INTERFACE I_Conveyor

PROPERTY bOccupied : BOOL
GET
END_GET
SET
END_SET
END_PROPERTY

PROPERTY eMode : E_ConveyorMode
GET
END_GET
SET
END_SET
END_PROPERTY

PROPERTY fCurrentSpeed : LREAL
GET
END_GET
SET
END_SET
END_PROPERTY

METHOD M_Divert : BOOL
VAR_INPUT
	bOpen : BOOL;
END_VAR
END_METHOD

METHOD M_reset : BOOL
VAR_INPUT
END_VAR
END_METHOD

METHOD M_run : BOOL
VAR_INPUT
	bForward : BOOL;
END_VAR
END_METHOD

METHOD M_Stop : BOOL
VAR_INPUT
END_VAR
END_METHOD

END_INTERFACE

(* stored: Version 1.1.0.1, ProductVersion 3.1.4024.16
   Itf I_Conveyor: Id {79695f05-cf47-4e8b-96fd-9364dffb9874}
   Property bOccupied: Id {c9acc93a-6b8f-48c7-a488-6008eeb0af8a}
   Get Get: Id {49011979-9998-412e-9dad-7bf1b1982af2}
   Set Set: Id {9cae3bd8-98bb-4139-b19e-d188c30ecd02}
   Property eMode: Id {b3a2cf31-50ff-4212-bb5d-f5315b579633}
   Get Get: Id {91cd94a6-8124-4b17-aa62-eef95d98fd70}
   Set Set: Id {6359936c-f76f-4018-9da6-0e0b9fb90406}
   Property fCurrentSpeed: Id {2380c4b5-8bda-4483-be69-9d50c0877aa3}
   Get Get: Id {9bc2dc8a-e6a9-4bbc-95ab-cee2ea1f471c}
   Set Set: Id {b3fbf38f-de76-41e7-a1e0-e0158ecbf0d7}
   Method M_Divert: Id {e45ca485-9837-4e48-bdfe-7ec21838192d}
   Method M_reset: Id {2c3869a7-9ecd-4f88-8df5-2c1fd23ea136}
   Method M_run: Id {9d109452-f5fe-4bde-932b-0963eea8677a}
   Method M_Stop: Id {4ad5a279-adc1-4e20-aa08-f54f49f7075c} *)
